// TIA Portal project "VENTILADORES" (V17)

(* hardware
DEVICE "S7-1500/ET200MP station_1"  S7-1500 station
   slot 0: "Rail_0"  Rack  6ES7 590-1***0-0AA0
   slot 1: "PLC_1"  CPU 1512C-1 PN  6ES7 512-1CK00-0AB0  V2.1
      slot 3: "CPU display_1"  6ES7591-1AA00-0AA0
      slot 32768: "PROFINET interface_1"  X1
         slot 32769: "Port_1"  X1 P1
         slot 32770: "Port_2"  X1 P2
*)

// ===== PLC "PLC_1"  CPU 1512C-1 PN =====

VAR_GLOBAL   // PLC tag table "Default tag table"
   "MARCA TEMPERATURA ADECUADA" AT %M0.0 : Bool;
   "MARCA TEMPERATURA INADECUADA FRIA" AT %M0.1 : Bool;
   "VENTILADOR M1" AT %Q0.0 : Bool;
   "VENTILADOR M2" AT %Q0.1 : Bool;
   "TEMPERATURA SALA" AT %ID0 : DInt;
   "TEMPERATURA DESEADA" AT %ID4 : DInt;
   "MARCA TEMPERATURA ADECUADA-2" AT %M0.7 : Bool;
   "MARCA TEMPERATURA INADECUADA FRIA-2" AT %M1.0 : Bool;
   "MARCA RESISTENCIA" AT %M1.1 : Bool;
   "RESISTENCIA" AT %Q0.2 : Bool;
   "MARCA TEMPERATURA INADECUADA CALIENTE" AT %M1.2 : Bool;
   "MARCA TEMPERATURA INADECUADA CALIENTE-2" AT %M1.3 : Bool;
   "VÁLVULA AGUA FRÍA" AT %Q0.3 : Bool;
   "MARCA AGUA FRÍA" AT %M1.4 : Bool;
   "CALCULO-VALOR" AT %QD0 : Real;
   "Tag_4" AT %MD100 : Real;
   "Tag_6" AT %MD500 : Real;
   "VALOR DIFERENCIA TEMPERATURA" AT %MD2000 : Real;
   "System_Byte" AT %MB1000 : Byte;
   "FirstScan" AT %M1000.0 : Bool;
   "DiagStatusUpdate" AT %M1000.1 : Bool;
   "AlwaysTRUE" AT %M1000.2 : Bool;
   "AlwaysFALSE" AT %M1000.3 : Bool;
   "Clock_Byte" AT %MB200 : Byte;
   "Clock_10Hz" AT %M200.0 : Bool;
   "Clock_5Hz" AT %M200.1 : Bool;
   "Clock_2.5Hz" AT %M200.2 : Bool;
   "Clock_2Hz" AT %M200.3 : Bool;
   "Clock_1.25Hz" AT %M200.4 : Bool;
   "Clock_1Hz" AT %M200.5 : Bool;
   "Clock_0.625Hz" AT %M200.6 : Bool;
   "Clock_0.5Hz" AT %M200.7 : Bool;
   "VALOR TEMPERATURA SALA" AT %MD300 : DInt;
END_VAR

DATA_BLOCK "PRUEBA"   // DB6
{ S7_Optimized_Access := 'FALSE' }
VERSION : 0.1
   VAR
      "TEMPERATURA SALA" : DInt := 10;
      "TEMPERATIRA DESEADA" : DInt := 20;
   END_VAR
BEGIN
END_DATA_BLOCK

FUNCTION "FC-SALIDAS" : Void   // FC1, LAD
{ S7_Optimized_Access := 'TRUE' }
VERSION : 0.1
BEGIN

REGION Network 1: VENTILADOR 1
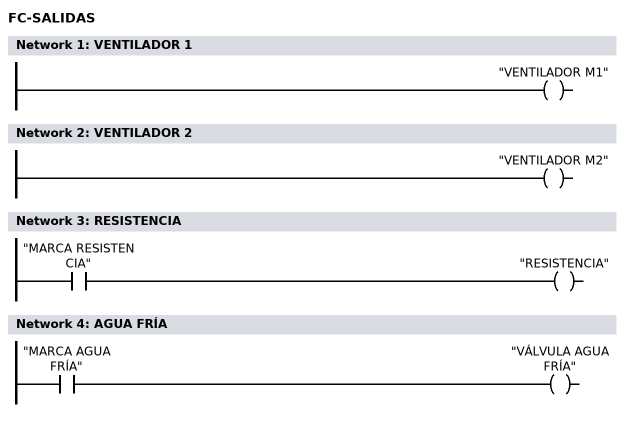
   RUNG wire#powerrail
      Coil( "VENTILADOR M1" )
   END_RUNG
   // the same network as SCL:
   "VENTILADOR M1" := TRUE;
END_REGION

REGION Network 2: VENTILADOR 2
   RUNG wire#powerrail
      Coil( "VENTILADOR M2" )
   END_RUNG
   // the same network as SCL:
   "VENTILADOR M2" := TRUE;
END_REGION

REGION Network 3: RESISTENCIA
   RUNG wire#powerrail
      Contact( "MARCA RESISTENCIA" )
      Coil( "RESISTENCIA" )
   END_RUNG
   // the same network as SCL:
   "RESISTENCIA" := "MARCA RESISTENCIA";
END_REGION

REGION Network 4: AGUA FRÍA
   RUNG wire#powerrail
      Contact( "MARCA AGUA FRÍA" )
      Coil( "VÁLVULA AGUA FRÍA" )
   END_RUNG
   // the same network as SCL:
   "VÁLVULA AGUA FRÍA" := "MARCA AGUA FRÍA";
END_REGION
END_FUNCTION

FUNCTION "FC-CONTROL" : Void   // FC2, LAD
{ S7_Optimized_Access := 'TRUE' }
VERSION : 0.1
BEGIN

REGION Network 1: MARCA RESISTENCIA
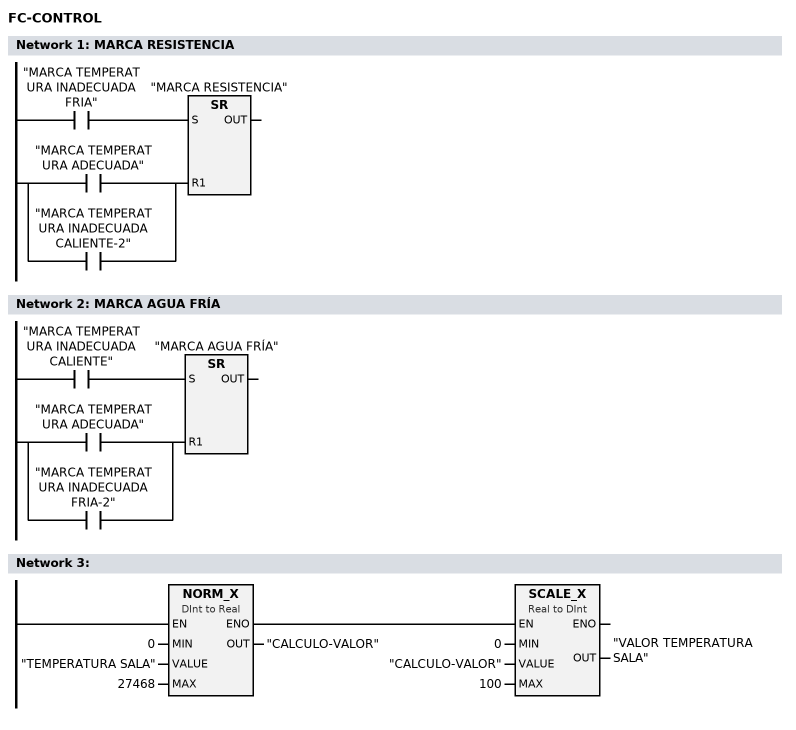
   RUNG wire#powerrail
      Contact( "MARCA TEMPERATURA INADECUADA FRIA" )
      S_SR(operand := "MARCA RESISTENCIA", r1 := wire#w1)
   END_RUNG
   RUNG wire#powerrail
      Contact( "MARCA TEMPERATURA ADECUADA" )
   END_RUNG wire#w1
   RUNG wire#powerrail
      Contact( "MARCA TEMPERATURA INADECUADA CALIENTE-2" )
   END_RUNG wire#w1
   // the same network as SCL:
   IF "MARCA TEMPERATURA INADECUADA FRIA" THEN
       "MARCA RESISTENCIA" := TRUE;   // SR flip-flop
   END_IF;
   IF "MARCA TEMPERATURA ADECUADA" OR "MARCA TEMPERATURA INADECUADA CALIENTE-2" THEN
       "MARCA RESISTENCIA" := FALSE;
   END_IF;
END_REGION

REGION Network 2: MARCA AGUA FRÍA
   RUNG wire#powerrail
      Contact( "MARCA TEMPERATURA INADECUADA CALIENTE" )
      S_SR(operand := "MARCA AGUA FRÍA", r1 := wire#w1)
   END_RUNG
   RUNG wire#powerrail
      Contact( "MARCA TEMPERATURA ADECUADA" )
   END_RUNG wire#w1
   RUNG wire#powerrail
      Contact( "MARCA TEMPERATURA INADECUADA FRIA-2" )
   END_RUNG wire#w1
   // the same network as SCL:
   IF "MARCA TEMPERATURA INADECUADA CALIENTE" THEN
       "MARCA AGUA FRÍA" := TRUE;   // SR flip-flop
   END_IF;
   IF "MARCA TEMPERATURA ADECUADA" OR "MARCA TEMPERATURA INADECUADA FRIA-2" THEN
       "MARCA AGUA FRÍA" := FALSE;
   END_IF;
END_REGION

REGION Network 3
   RUNG wire#powerrail
      { S7_Templates := "[SrcType := DInt, DestType := Real]" } Normalize(min := 0, value := "TEMPERATURA SALA", max := 27468, out => "CALCULO-VALOR")
      { S7_Templates := "[SrcType := Real, DestType := DInt]" } Scale(min := 0, value := "CALCULO-VALOR", max := 100, out => "VALOR TEMPERATURA SALA")
   END_RUNG
   // the same network as SCL:
   "CALCULO-VALOR" := NORM_X(MIN := 0, VALUE := "TEMPERATURA SALA", MAX := 27468);
   "VALOR TEMPERATURA SALA" := SCALE_X(MIN := 0, VALUE := "CALCULO-VALOR", MAX := 100);
END_REGION
END_FUNCTION

FUNCTION "FC-SECUENCIA" : Void   // FC3, LAD
{ S7_Optimized_Access := 'TRUE' }
VERSION : 0.1
BEGIN

REGION Network 1: TEMPERATURA ADECUADA
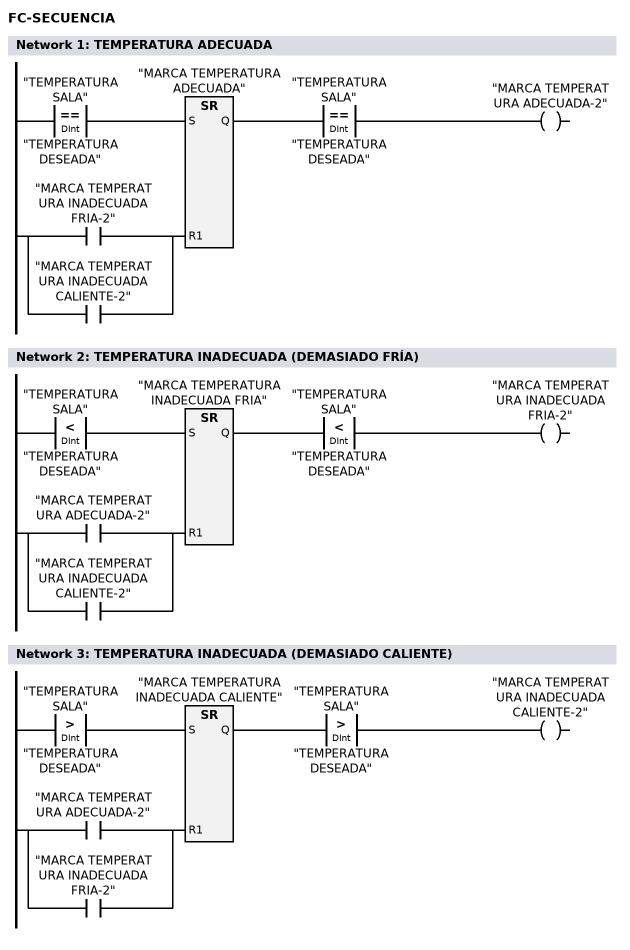
   RUNG wire#powerrail
      { S7_Templates := "SrcType := DInt" } EQ_Contact(in1 := "TEMPERATURA SALA", in2 := "TEMPERATURA DESEADA")
      S_SR(operand := "MARCA TEMPERATURA ADECUADA", r1 := wire#w1)
      { S7_Templates := "SrcType := DInt" } EQ_Contact(in1 := "TEMPERATURA SALA", in2 := "TEMPERATURA DESEADA")
      Coil( "MARCA TEMPERATURA ADECUADA-2" )
   END_RUNG
   RUNG wire#powerrail
      Contact( "MARCA TEMPERATURA INADECUADA FRIA-2" )
   END_RUNG wire#w1
   RUNG wire#powerrail
      Contact( "MARCA TEMPERATURA INADECUADA CALIENTE-2" )
   END_RUNG wire#w1
   // the same network as SCL:
   IF "TEMPERATURA SALA" = "TEMPERATURA DESEADA" THEN
       "MARCA TEMPERATURA ADECUADA" := TRUE;   // SR flip-flop
   END_IF;
   IF "MARCA TEMPERATURA INADECUADA FRIA-2" OR "MARCA TEMPERATURA INADECUADA CALIENTE-2" THEN
       "MARCA TEMPERATURA ADECUADA" := FALSE;
   END_IF;
   "MARCA TEMPERATURA ADECUADA-2" := "MARCA TEMPERATURA ADECUADA" AND ("TEMPERATURA SALA" = "TEMPERATURA DESEADA");
END_REGION

REGION Network 2: TEMPERATURA INADECUADA (DEMASIADO FRÍA)
   RUNG wire#powerrail
      { S7_Templates := "SrcType := DInt" } LT_Contact(in1 := "TEMPERATURA SALA", in2 := "TEMPERATURA DESEADA")
      S_SR(operand := "MARCA TEMPERATURA INADECUADA FRIA", r1 := wire#w1)
      { S7_Templates := "SrcType := DInt" } LT_Contact(in1 := "TEMPERATURA SALA", in2 := "TEMPERATURA DESEADA")
      Coil( "MARCA TEMPERATURA INADECUADA FRIA-2" )
   END_RUNG
   RUNG wire#powerrail
      Contact( "MARCA TEMPERATURA ADECUADA-2" )
   END_RUNG wire#w1
   RUNG wire#powerrail
      Contact( "MARCA TEMPERATURA INADECUADA CALIENTE-2" )
   END_RUNG wire#w1
   // the same network as SCL:
   IF "TEMPERATURA SALA" < "TEMPERATURA DESEADA" THEN
       "MARCA TEMPERATURA INADECUADA FRIA" := TRUE;   // SR flip-flop
   END_IF;
   IF "MARCA TEMPERATURA ADECUADA-2" OR "MARCA TEMPERATURA INADECUADA CALIENTE-2" THEN
       "MARCA TEMPERATURA INADECUADA FRIA" := FALSE;
   END_IF;
   "MARCA TEMPERATURA INADECUADA FRIA-2" := "MARCA TEMPERATURA INADECUADA FRIA" AND ("TEMPERATURA SALA" < "TEMPERATURA DESEADA");
END_REGION

REGION Network 3: TEMPERATURA INADECUADA (DEMASIADO CALIENTE)
   RUNG wire#powerrail
      { S7_Templates := "SrcType := DInt" } GT_Contact(in1 := "TEMPERATURA SALA", in2 := "TEMPERATURA DESEADA")
      S_SR(operand := "MARCA TEMPERATURA INADECUADA CALIENTE", r1 := wire#w1)
      { S7_Templates := "SrcType := DInt" } GT_Contact(in1 := "TEMPERATURA SALA", in2 := "TEMPERATURA DESEADA")
      Coil( "MARCA TEMPERATURA INADECUADA CALIENTE-2" )
   END_RUNG
   RUNG wire#powerrail
      Contact( "MARCA TEMPERATURA ADECUADA-2" )
   END_RUNG wire#w1
   RUNG wire#powerrail
      Contact( "MARCA TEMPERATURA INADECUADA FRIA-2" )
   END_RUNG wire#w1
   // the same network as SCL:
   IF "TEMPERATURA SALA" > "TEMPERATURA DESEADA" THEN
       "MARCA TEMPERATURA INADECUADA CALIENTE" := TRUE;   // SR flip-flop
   END_IF;
   IF "MARCA TEMPERATURA ADECUADA-2" OR "MARCA TEMPERATURA INADECUADA FRIA-2" THEN
       "MARCA TEMPERATURA INADECUADA CALIENTE" := FALSE;
   END_IF;
   "MARCA TEMPERATURA INADECUADA CALIENTE-2" := "MARCA TEMPERATURA INADECUADA CALIENTE" AND ("TEMPERATURA SALA" > "TEMPERATURA DESEADA");
END_REGION
END_FUNCTION

FUNCTION "FC-TEMPERATURA" : Void   // FC4, SCL
{ S7_Optimized_Access := 'TRUE' }
VERSION : 0.1
BEGIN
   IF "TEMPERATURA SALA" > "TEMPERATURA DESEADA" THEN
       "MARCA AGUA FRÍA" := 1;
       "MARCA RESISTENCIA" := 0;
   ELSIF"TEMPERATURA SALA" < "TEMPERATURA DESEADA" THEN
       "MARCA RESISTENCIA" := 1;
       "MARCA AGUA FRÍA" := 0;
   ELSE
       "MARCA AGUA FRÍA" := 0;
       "MARCA RESISTENCIA" := 0;
   END_IF;
END_FUNCTION

ORGANIZATION_BLOCK "Main"   // OB1, LAD, ProgramCycle
TITLE = "Main Program Sweep (Cycle)"
{ S7_Optimized_Access := 'TRUE' }
VERSION : 0.1
   VAR_INPUT
      Initial_Call : Bool;   // Initial call of this OB
      Remanence : Bool;   // =True, if remanent data are available
   END_VAR
BEGIN

REGION Network 1
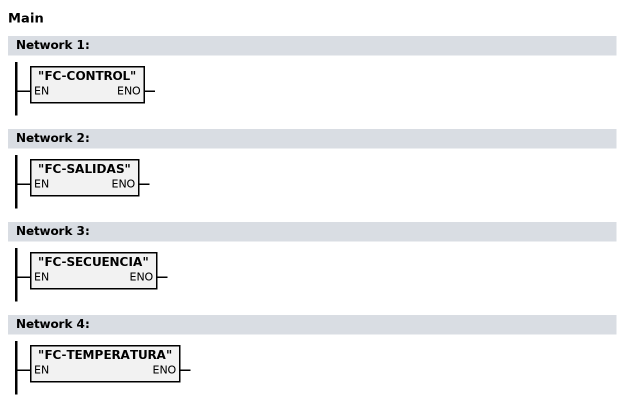
   RUNG wire#powerrail
      "FC-CONTROL"()
   END_RUNG
   // the same network as SCL:
   "FC-CONTROL"();
END_REGION

REGION Network 2
   RUNG wire#powerrail
      "FC-SALIDAS"()
   END_RUNG
   // the same network as SCL:
   "FC-SALIDAS"();
END_REGION

REGION Network 3
   RUNG wire#powerrail
      "FC-SECUENCIA"()
   END_RUNG
   // the same network as SCL:
   "FC-SECUENCIA"();
END_REGION

REGION Network 4
   RUNG wire#powerrail
      "FC-TEMPERATURA"()
   END_RUNG
   // the same network as SCL:
   "FC-TEMPERATURA"();
END_REGION
END_ORGANIZATION_BLOCK

ORGANIZATION_BLOCK "OB30"   // OB30, LAD, CyclicInterrupt
{ S7_Optimized_Access := 'TRUE' }
VERSION : 0.1
   VAR_INPUT
      Initial_Call : Bool;   // Initial call of this OB
      Event_Count : Int;   // Events discarded
   END_VAR
BEGIN

REGION Network 1
   // ME DA EL VALOR (EN %) DE LA DIFERENCIA QUE HAY ENTRE EL INPUT Y EL SETPOINT (SP)
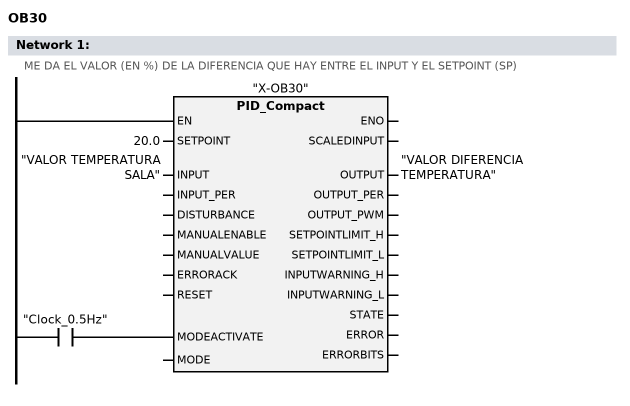
   "X-OB30"(Setpoint := 20.0,   // PID_Compact
            Input := "VALOR TEMPERATURA SALA",
            ModeActivate := "Clock_0.5Hz",
            Output => "VALOR DIFERENCIA TEMPERATURA");
END_REGION
END_ORGANIZATION_BLOCK